TYPE csp_case_flap_control_status_enum :
(
	CSP_CASE_FLAP_CONTROL_STATUS_NOT_INITIALIZED 							:=  0,
	CSP_CASE_FLAP_CONTROL_STATUS_DISABLED 									:=  10,
	CSP_CASE_FLAP_CONTROL_STATUS_ENABLE_REQUEST 							:=  20,
	CSP_CASE_FLAP_CONTROL_STATUS_ENABLING 									:=  30,
	CSP_CASE_FLAP_CONTROL_STATUS_ENABLED 									:=  40,
	CSP_CASE_FLAP_CONTROL_STATUS_CHANGE_OVER_MODE							:=  45,
	CSP_CASE_FLAP_CONTROL_STATUS_CHANGE_OVER_MODE_DONE						:= 	47,
	CSP_CASE_FLAP_CONTROL_STATUS_HOME_REQUEST								:=  50,
	CSP_CASE_FLAP_CONTROL_STATUS_HOMING										:=  60,
	CSP_CASE_FLAP_CONTROL_STATUS_HOME_DONE									:=  70,
	CSP_CASE_FLAP_CONTROL_STATUS_CALCULATING_SLAVE_POSITION					:=  90,
	CSP_CASE_FLAP_CONTROL_STATUS_WAITING_SLAVE_ENGAGE						:= 100,
	CSP_CASE_FLAP_CONTROL_STATUS_WAITING_SLAVE_ENGAGE_2						:= 120,
	CSP_CASE_FLAP_CONTROL_STATUS_PHASE_REQUEST								:= 140,
	CSP_CASE_FLAP_CONTROL_STATUS_PHASING									:= 150,
	CSP_CASE_FLAP_CONTROL_STATUS_PHASED										:= 160,
	CSP_CASE_FLAP_CONTROL_STATUS_CAM_ENGAGED_REQ							:= 170,
	CSP_CASE_FLAP_CONTROL_STATUS_AXIS_ENGAGE_VERIFY							:= 180,
	CSP_CASE_FLAP_CONTROL_STATUS_CAM_ENGAGED								:= 190,
	CSP_CASE_FLAP_CONTROL_STATUS_CAM_TABLE_READ								:= 195,
	CSP_CASE_FLAP_CONTROL_STATUS_CALCULATE_SLAVE_POSITION_REQUEST			:= 196,
	CSP_CASE_FLAP_CONTROL_STATUS_READY										:= 197,
	CSP_CASE_FLAP_CONTROL_STATUS_RUNNING									:= 200,
	CSP_CASE_FLAP_CONTROL_STATUS_MOVING										:= 205,
	CSP_CASE_FLAP_CONTROL_STATUS_DISENGAGE_REQUEST							:= 210,
	CSP_CASE_FLAP_CONTROL_STATUS_DISENGAGING								:= 211,	
	
	
	CSP_CASE_FLAP_CONTROL_STATUS_STOP_REQUEST 								:= 500,
	CSP_CASE_FLAP_CONTROL_STATUS_DISABLE_REQUEST 							:= 530,
	CSP_CASE_FLAP_CONTROL_STATUS_DISABLING 									:= 540
) := CSP_CASE_FLAP_CONTROL_STATUS_NOT_INITIALIZED;
END_TYPE

(* stored: Version 1.1.0.1, ProductVersion 3.1.4024.3
   DUT csp_case_flap_control_status_enum: Id {32f7e41c-e30c-4819-ac27-926b03cbd7e8} *)
